(*
 * Contains every service relevant to Resi4MPM control.
 * Used so that the services can use each other (similar to dependency injection).
 *)
FUNCTION_BLOCK ServiceContainer
VAR_INPUT
END_VAR
VAR_OUTPUT
END_VAR
VAR
	m_ptrErrorMgr: POINTER TO ErrorManagerBase;
	
	m_pm: ProcessManager;
	m_ptrProcessManager: POINTER TO ProcessManager := ADR(m_pm);
 
	m_st: StateTracker;
	m_ptrStateTracker: POINTER TO StateTracker := ADR(m_st);
END_VAR

METHOD FB_init : BOOL
VAR_INPUT
	bInitRetains : BOOL; // if TRUE, the retain variables are initialized (warm start / cold start)
	bInCopyCode : BOOL;  // if TRUE, the instance afterwards gets moved into the copy code (online change)
	
	i_ptrErrorMgr: POINTER TO ErrorManagerBase;
END_VAR
// get the APPLICATION-SPECIFIC services
THIS^.m_ptrErrorMgr := i_ptrErrorMgr;

// initialize all services
THIS^.m_ptrProcessManager^.ProvideServices(THIS^.m_ptrStateTracker, i_ptrErrorMgr);
THIS^.m_ptrStateTracker^.ProvideServices(THIS^.m_ptrProcessManager, i_ptrErrorMgr);
END_METHOD

PROPERTY PtrErrorManager : POINTER TO ErrorManagerBase
GET
PtrErrorManager := m_ptrErrorMgr;
END_GET
END_PROPERTY

PROPERTY PtrProcessManager : POINTER TO ProcessManager
GET
PtrProcessManager := THIS^.m_ptrProcessManager;
END_GET
END_PROPERTY

PROPERTY PtrStateTracker : POINTER TO StateTracker
GET
PtrStateTracker := THIS^.m_ptrStateTracker;
END_GET
END_PROPERTY

END_FUNCTION_BLOCK

(* stored: Version 1.1.0.1
   POU ServiceContainer: Id {d47a98b4-53a9-4c2d-91de-97e499d45816}, SpecialFunc None
   Method FB_init: Id {76b2eb79-139b-460f-9d2b-c3c8fec35c9a}
   Property PtrErrorManager: Id {bcbb9720-c928-4528-b39f-6343631f28e9}
   Get Get: Id {5d953ccd-6d3e-447f-8101-0260ac0bc9f0}
   Property PtrProcessManager: Id {abf72391-ab31-45bb-8183-a763441ec63a}
   Get Get: Id {0cc721ff-faa8-4a61-9b3e-b94adb1dcc72}
   Property PtrStateTracker: Id {d493ebf2-eab6-4511-b2e2-e5ddce193eb4}
   Get Get: Id {e380312d-47f7-457c-abb6-e2a1bbfd4fac} *)
